// SIMATIC S7-200 project (STEP 7-Micro/WIN), CPU 221 REL 01.10

SYMBOL_TABLE USER1
K                Q0.0     // PISTONG
S1               I0.0     // cho pistong chay ra
S2               I0.1     // cho pistong rut vao
END_SYMBOL_TABLE

ORGANIZATION_BLOCK MAIN:OB1
TITLE=nhan start pistong chay ra 5s sau pistong chay vao
BEGIN
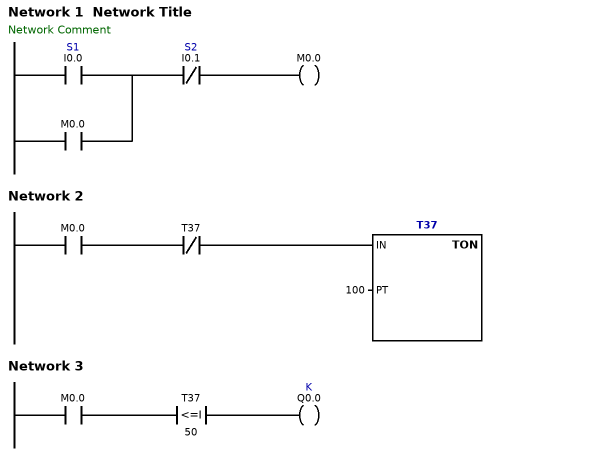
Network 1 // Network Title
// Network Comment
LD     S1:I0.0
O      M0.0
AN     S2:I0.1
=      M0.0
Network 2
LD     M0.0
AN     T37
TON    T37, 100
Network 3
LD     M0.0
AW<=   T37, 50
=      K:Q0.0
END_ORGANIZATION_BLOCK
